{attribute 'GeneratedUsingTerminal: EPP1342-0001-0016'}
{attribute addProperty BoxType "EPP1342-0001-0016"}
{attribute addProperty Id "A_0024_EPP1342_0001_0017A_0024_EPP1342_0001_0017_01FF1674322"}
{attribute addProperty CRC "1700668326"}
{attribute addProperty Size "322"}
TYPE A_0023_EPP1342_0001_0016_655E23A6 EXTENDS EPP1342_1FC0878B :
STRUCT
	{attribute addProperty Name "A_0024_EPP1342_0001_0017"}
	{attribute addProperty PreviousPort "A_0023(EPP1342-0001-0016) : D"}
	A_0024_EPP1342_0001_0017 : A_0024_EPP1342_0001_0017_01FF1674;
END_STRUCT
END_TYPE

(* stored: Version 1.2.0.0, ProductVersion 3.1.4024.9
   DUT A_0023_EPP1342_0001_0016_655E23A6: Id {40858f47-a28d-49b7-a479-9e7627aaac6f} *)
